Fanuc KAREL source: worienttype.kl

PROGRAM worienttype
%NOLOCKGROUP
VAR
  p : POSITION
  q : POSITION
  i : INTEGER
  r : REAL
BEGIN
  WITH $ORIENT_TYPE = RSWORLD MOVE TO p
END worienttype
